PROGRAM main
  VAR
    ProductSensor : BOOL;
    ResetBtn : BOOL;
    ConveyorMotor : BOOL;
    BoxFull : BOOL;
    CTU0 : CTU;
  END_VAR

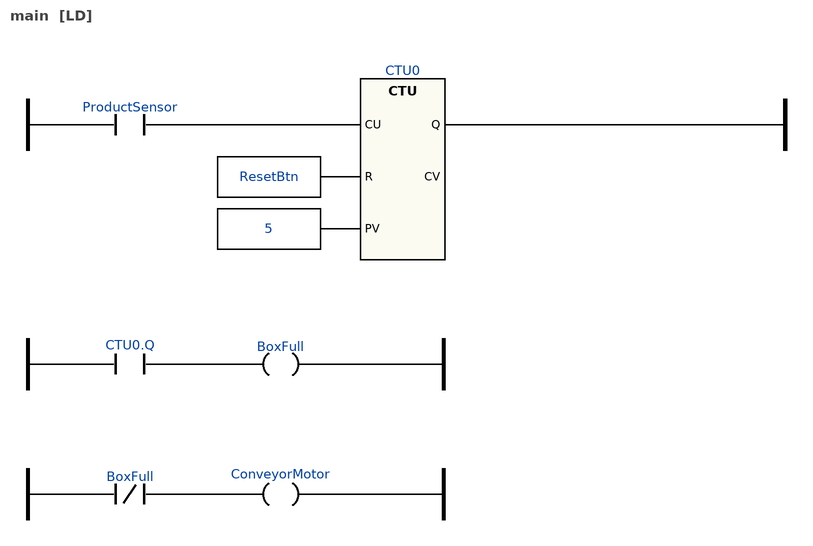
(* LD diagram, written out as Structured Text *)
BoxFull := CTU0.Q;
ConveyorMotor := NOT BoxFull;
CTU0(CU := ProductSensor, R := ResetBtn, PV := 5);
END_PROGRAM
